(* CODESYS project Agitator.xml

Project tree, tasks and I/O mapping:
  function block Agitator [LD]
*)

// Agitator
FUNCTION_BLOCK Agitator
// The Agitator function block is for managing the agitator in the hopper.
// The agitator needs to run a agitator "cycle", called the agitator sequence, periodically to make sure 
// the ice doesn't stick together. The agitator also runs while feeding ice, and stirs the ice when full 
// to make sure there aren't any voids in the hopper making you think the hopper is totally full.
VAR_INPUT
	Enable: 			BOOL;
	ManualAgitate: 		BOOL; 				// A bit to manually agitate, controlled from an HMI button exposed for maintenance functionality.
	StirIce: 			BOOL; 				// A bit to manually agitate after reaching the max sensor.
	FeedIce: 			BOOL; 				// A bit to run the agitator when feeding ice.
	AutoAgitate: 		BOOL; 				// A bit to activate auto agitating cycle.
	ReverseTime: 		TIME; 				// Agitator cycle time spent in reverse motion.
	DwellTime: 			TIME;   			// Agitator cycle time spent dwelling between reverse-forward motion.
	ForwardTime: 		TIME; 				// Agitator cycle time spent in forward motion.
	IdleTime: 			TIME;    			// Time spent idling between automatic agitator cycles.
END_VAR
VAR_OUTPUT
	Agitating: 			BOOL; 				// A helper bit to indicate agitating is active.
	Forward: 			BOOL; 				// Agitator motor VFD forward.
	Reverse: 			BOOL; 				// Agitator motor VFD reverse.
	CycleComplete: 		BOOL; 				// A bit that pulses everytime an agitate cycle completes.
	SinceLastAgitate: 	TIME; 				// Time since the last agitate cycle completed.
END_VAR
VAR
	_RunForward: 		BOOL;
	_RunReverse: 		BOOL;
	_Dwell: 			BOOL;
	_Trigger: 			BOOL;
	_Sequence: 			AgitatorSequence;
	_IdleTimer: 		TON;
	_CompleteTimer: 	TOF;
END_VAR
VAR // added by the converter: edge detectors and wires of the graphical bodies
    _rt1 : R_TRIG;
END_VAR

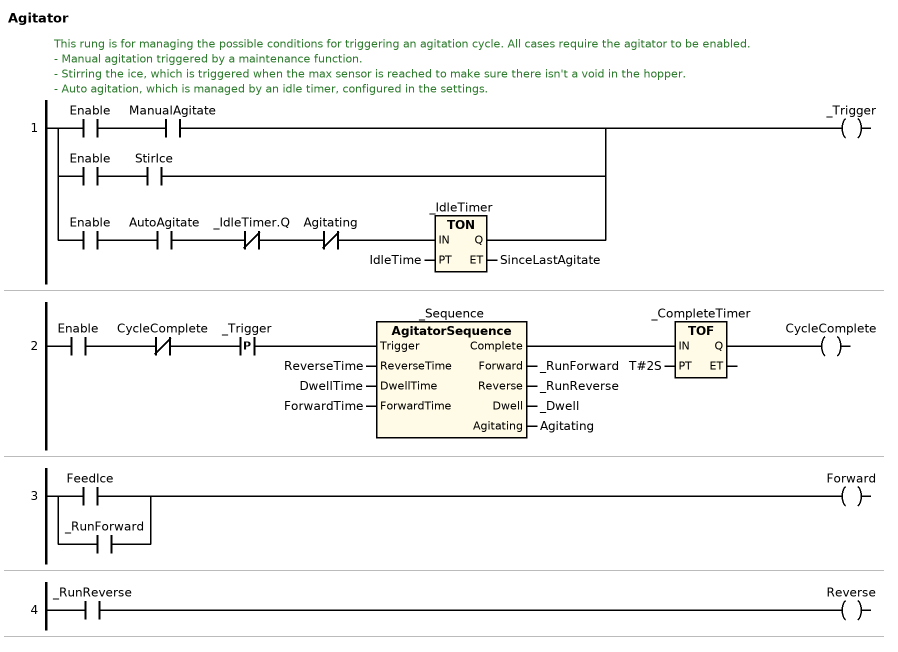
// NETWORK 1
// This rung is for managing the possible conditions for triggering an agitation cycle. All cases require the agitator to be enabled.
//  - Manual agitation triggered by a maintenance function.
//  - Stirring the ice, which is triggered when the max sensor is reached to make sure there isn't a void in the hopper.
//  - Auto agitation, which is managed by an idle timer, configured in the settings.
_IdleTimer(
    IN := Enable AND AutoAgitate AND NOT _IdleTimer.Q AND NOT Agitating,
    PT := IdleTime,
    ET => SinceLastAgitate); // TON
_Trigger := Enable AND ManualAgitate OR Enable AND StirIce OR _IdleTimer.Q;

// NETWORK 2
_rt1(CLK := _Trigger);
_Sequence(
    Trigger := Enable AND NOT CycleComplete AND _rt1.Q,
    ReverseTime := ReverseTime,
    DwellTime := DwellTime,
    ForwardTime := ForwardTime,
    Forward => _RunForward,
    Reverse => _RunReverse,
    Dwell => _Dwell,
    Agitating => Agitating); // AgitatorSequence
_CompleteTimer(IN := _Sequence.Complete, PT := T#2S); // TOF
CycleComplete := _CompleteTimer.Q;

// NETWORK 3
Forward := FeedIce OR _RunForward;

// NETWORK 4
Reverse := _RunReverse;

END_FUNCTION_BLOCK
